// TIA Portal V17 export
// export: Created 2026-04-12T10:31:28.5302505Z, ExportSetting WithDefaults, DisplayName Totally Integrated Automation Portal, DisplayVersion V17 Update 4, DisplayName TIA Portal Openness, DisplayVersion V17 Update 4, DisplayName TIA Portal Version Control Interface, DisplayVersion V17, DisplayName SINAMICS Startdrive Advanced, DisplayVersion V17, DisplayName SINAMICS Startdrive G130, G150, S120, S150, SINAMICS MV, S210, DisplayVersion V17, DisplayName SINAMICS Startdrive G110M, G120, G120C, G120D, G120P, G115D, DisplayVersion V17, DisplayName STEP 7 Professional, DisplayVersion V17 Update 4, DisplayName STEP 7 Safety, DisplayVersion V17, DisplayName WinCC Advanced, DisplayVersion V17 Update 4
FUNCTION "设定值传递" : Void   // FC1, LAD
{ S7_Optimized_Access := 'TRUE' }
VERSION : 0.1
// stored: AutoNumber false, IsIECCheckEnabled false, SetENOAutomatically false, UDAEnableTagReadback false
   VAR_TEMP   // added for the SCL form of the ladder/FBD networks
      _w1 : Bool;
      _w2 : Bool;
   END_VAR
BEGIN

REGION Network 1: 程序停止时
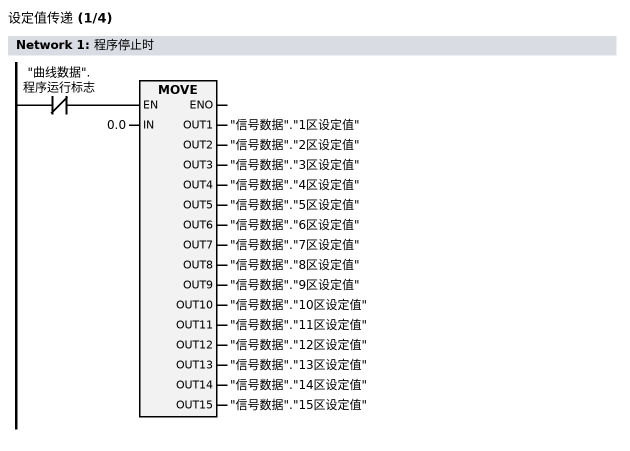
   RUNG wire#powerrail
      I_Contact( "曲线数据".程序运行标志 )
      Move(in := 0.0, out1 => "信号数据"."1区设定值", out2 => "信号数据"."2区设定值", out3 => "信号数据"."3区设定值", out4 => "信号数据"."4区设定值", out5 => "信号数据"."5区设定值", out6 => "信号数据"."6区设定值", out7 => "信号数据"."7区设定值", out8 => "信号数据"."8区设定值", out9 => "信号数据"."9区设定值", out10 => "信号数据"."10区设定值", out11 => "信号数据"."11区设定值", out12 => "信号数据"."12区设定值", out13 => "信号数据"."13区设定值", out14 => "信号数据"."14区设定值", out15 => "信号数据"."15区设定值")
   END_RUNG
   // the same network as SCL:
   IF NOT "曲线数据".程序运行标志 THEN
       "信号数据"."1区设定值" := 0.0;
       "信号数据"."2区设定值" := 0.0;
       "信号数据"."3区设定值" := 0.0;
       "信号数据"."4区设定值" := 0.0;
       "信号数据"."5区设定值" := 0.0;
       "信号数据"."6区设定值" := 0.0;
       "信号数据"."7区设定值" := 0.0;
       "信号数据"."8区设定值" := 0.0;
       "信号数据"."9区设定值" := 0.0;
       "信号数据"."10区设定值" := 0.0;
       "信号数据"."11区设定值" := 0.0;
       "信号数据"."12区设定值" := 0.0;
       "信号数据"."13区设定值" := 0.0;
       "信号数据"."14区设定值" := 0.0;
       "信号数据"."15区设定值" := 0.0;
   END_IF;
END_REGION

REGION Network 2: 程序运行但未暂停时
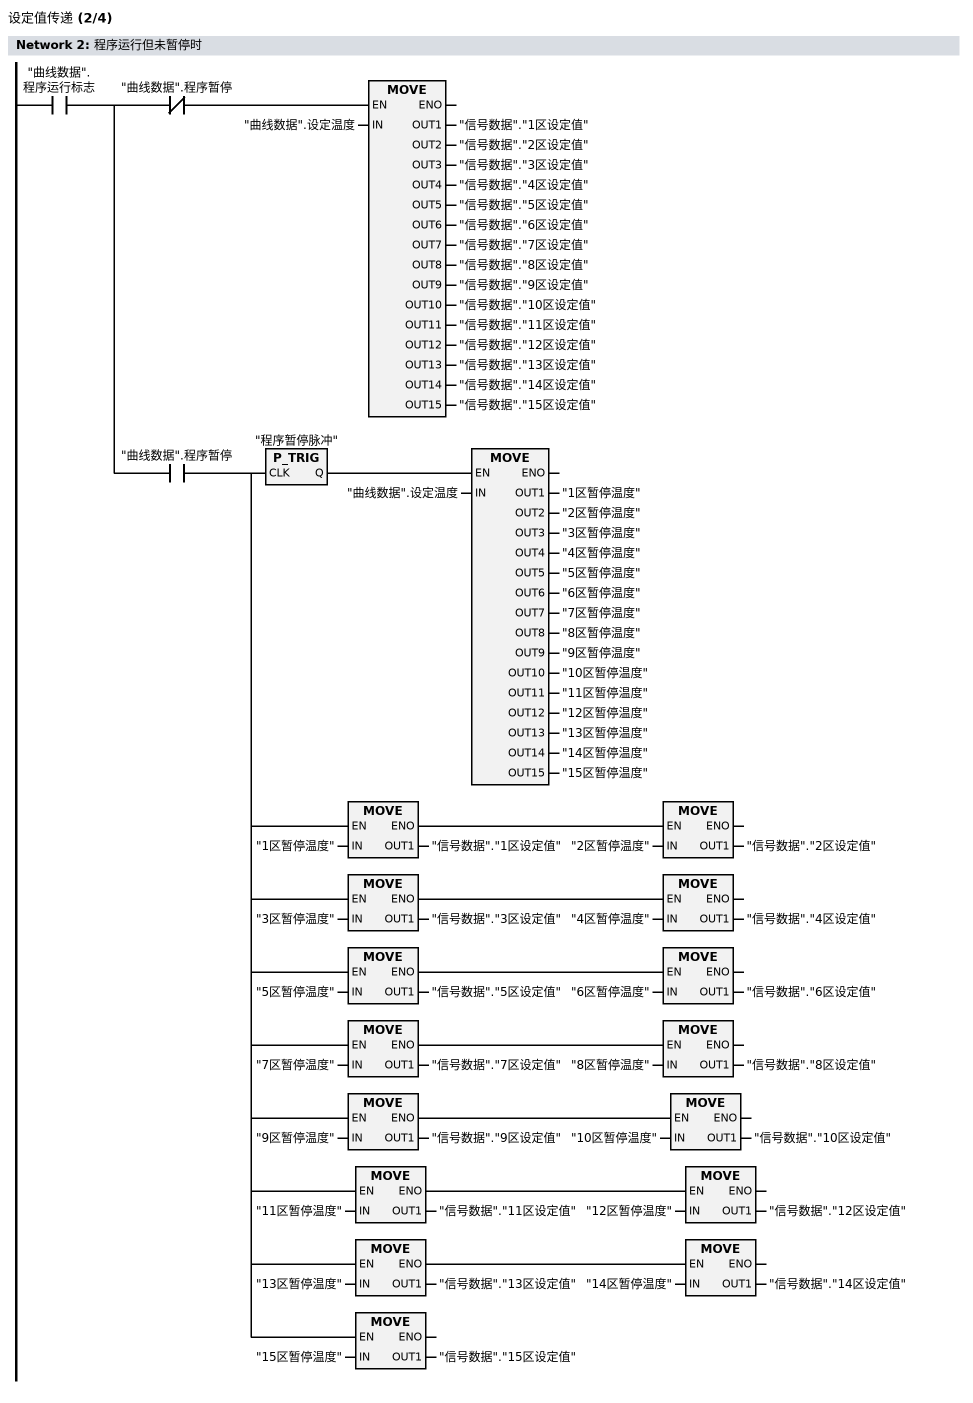
   RUNG wire#powerrail
      Contact( "曲线数据".程序运行标志 )
      wire#w1
      I_Contact( "曲线数据".程序暂停 )
      Move(in := "曲线数据".设定温度, out1 => "信号数据"."1区设定值", out2 => "信号数据"."2区设定值", out3 => "信号数据"."3区设定值", out4 => "信号数据"."4区设定值", out5 => "信号数据"."5区设定值", out6 => "信号数据"."6区设定值", out7 => "信号数据"."7区设定值", out8 => "信号数据"."8区设定值", out9 => "信号数据"."9区设定值", out10 => "信号数据"."10区设定值", out11 => "信号数据"."11区设定值", out12 => "信号数据"."12区设定值", out13 => "信号数据"."13区设定值", out14 => "信号数据"."14区设定值", out15 => "信号数据"."15区设定值")
   END_RUNG
   RUNG wire#w1
      Contact( "曲线数据".程序暂停 )
      wire#w2
      P_Trig( "程序暂停脉冲" )
      Move(in := "曲线数据".设定温度, out1 => "1区暂停温度", out2 => "2区暂停温度", out3 => "3区暂停温度", out4 => "4区暂停温度", out5 => "5区暂停温度", out6 => "6区暂停温度", out7 => "7区暂停温度", out8 => "8区暂停温度", out9 => "9区暂停温度", out10 => "10区暂停温度", out11 => "11区暂停温度", out12 => "12区暂停温度", out13 => "13区暂停温度", out14 => "14区暂停温度", out15 => "15区暂停温度")
   END_RUNG
   RUNG wire#w2
      Move(in := "1区暂停温度", out1 => "信号数据"."1区设定值")
      Move(in := "2区暂停温度", out1 => "信号数据"."2区设定值")
   END_RUNG
   RUNG wire#w2
      Move(in := "3区暂停温度", out1 => "信号数据"."3区设定值")
      Move(in := "4区暂停温度", out1 => "信号数据"."4区设定值")
   END_RUNG
   RUNG wire#w2
      Move(in := "5区暂停温度", out1 => "信号数据"."5区设定值")
      Move(in := "6区暂停温度", out1 => "信号数据"."6区设定值")
   END_RUNG
   RUNG wire#w2
      Move(in := "7区暂停温度", out1 => "信号数据"."7区设定值")
      Move(in := "8区暂停温度", out1 => "信号数据"."8区设定值")
   END_RUNG
   RUNG wire#w2
      Move(in := "9区暂停温度", out1 => "信号数据"."9区设定值")
      Move(in := "10区暂停温度", out1 => "信号数据"."10区设定值")
   END_RUNG
   RUNG wire#w2
      Move(in := "11区暂停温度", out1 => "信号数据"."11区设定值")
      Move(in := "12区暂停温度", out1 => "信号数据"."12区设定值")
   END_RUNG
   RUNG wire#w2
      Move(in := "13区暂停温度", out1 => "信号数据"."13区设定值")
      Move(in := "14区暂停温度", out1 => "信号数据"."14区设定值")
   END_RUNG
   RUNG wire#w2
      Move(in := "15区暂停温度", out1 => "信号数据"."15区设定值")
   END_RUNG
   // the same network as SCL:
   IF "曲线数据".程序运行标志 AND NOT "曲线数据".程序暂停 THEN
       "信号数据"."1区设定值" := "曲线数据".设定温度;
       "信号数据"."2区设定值" := "曲线数据".设定温度;
       "信号数据"."3区设定值" := "曲线数据".设定温度;
       "信号数据"."4区设定值" := "曲线数据".设定温度;
       "信号数据"."5区设定值" := "曲线数据".设定温度;
       "信号数据"."6区设定值" := "曲线数据".设定温度;
       "信号数据"."7区设定值" := "曲线数据".设定温度;
       "信号数据"."8区设定值" := "曲线数据".设定温度;
       "信号数据"."9区设定值" := "曲线数据".设定温度;
       "信号数据"."10区设定值" := "曲线数据".设定温度;
       "信号数据"."11区设定值" := "曲线数据".设定温度;
       "信号数据"."12区设定值" := "曲线数据".设定温度;
       "信号数据"."13区设定值" := "曲线数据".设定温度;
       "信号数据"."14区设定值" := "曲线数据".设定温度;
       "信号数据"."15区设定值" := "曲线数据".设定温度;
   END_IF;
   #_w1 := "曲线数据".程序运行标志 AND "曲线数据".程序暂停;
   #_w2 := #_w1 AND NOT "程序暂停脉冲";   // rising edge
   "程序暂停脉冲" := #_w1;
   IF #_w2 THEN
       "1区暂停温度" := "曲线数据".设定温度;
       "2区暂停温度" := "曲线数据".设定温度;
       "3区暂停温度" := "曲线数据".设定温度;
       "4区暂停温度" := "曲线数据".设定温度;
       "5区暂停温度" := "曲线数据".设定温度;
       "6区暂停温度" := "曲线数据".设定温度;
       "7区暂停温度" := "曲线数据".设定温度;
       "8区暂停温度" := "曲线数据".设定温度;
       "9区暂停温度" := "曲线数据".设定温度;
       "10区暂停温度" := "曲线数据".设定温度;
       "11区暂停温度" := "曲线数据".设定温度;
       "12区暂停温度" := "曲线数据".设定温度;
       "13区暂停温度" := "曲线数据".设定温度;
       "14区暂停温度" := "曲线数据".设定温度;
       "15区暂停温度" := "曲线数据".设定温度;
   END_IF;
   IF #_w1 THEN
       "信号数据"."1区设定值" := "1区暂停温度";
       "信号数据"."2区设定值" := "2区暂停温度";
       "信号数据"."3区设定值" := "3区暂停温度";
       "信号数据"."4区设定值" := "4区暂停温度";
       "信号数据"."5区设定值" := "5区暂停温度";
       "信号数据"."6区设定值" := "6区暂停温度";
       "信号数据"."7区设定值" := "7区暂停温度";
       "信号数据"."8区设定值" := "8区暂停温度";
       "信号数据"."9区设定值" := "9区暂停温度";
       "信号数据"."10区设定值" := "10区暂停温度";
       "信号数据"."11区设定值" := "11区暂停温度";
       "信号数据"."12区设定值" := "12区暂停温度";
       "信号数据"."13区设定值" := "13区暂停温度";
       "信号数据"."14区设定值" := "14区暂停温度";
       "信号数据"."15区设定值" := "15区暂停温度";
   END_IF;
END_REGION

REGION Network 3: 程序运行瞬间复位自动
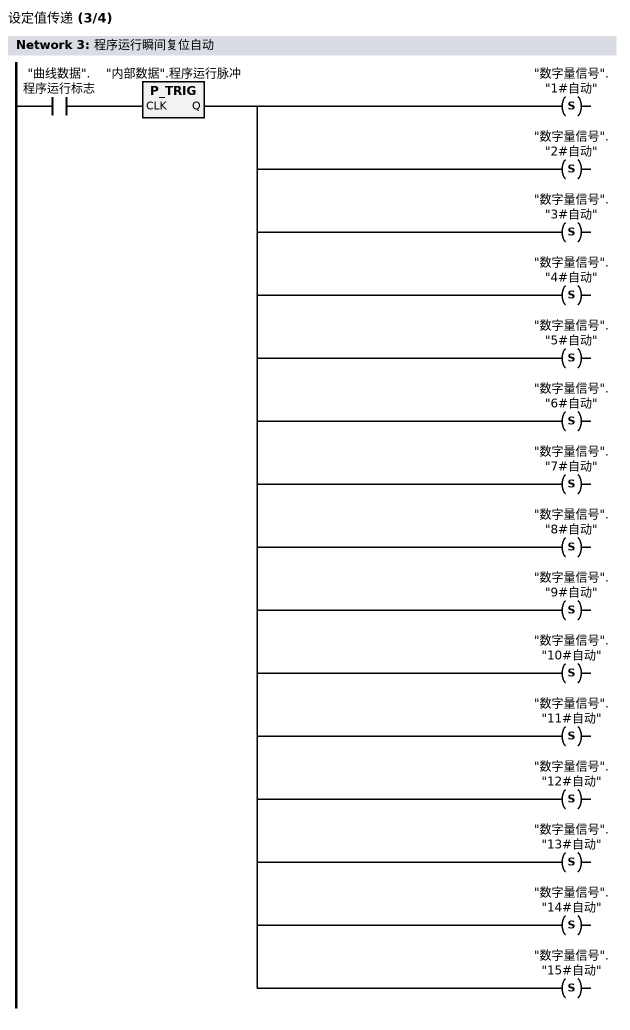
   RUNG wire#powerrail
      Contact( "曲线数据".程序运行标志 )
      P_Trig( "内部数据".程序运行脉冲 )
      wire#w1
      S_Coil( "数字量信号"."1#自动" )
   END_RUNG
   RUNG wire#w1
      S_Coil( "数字量信号"."2#自动" )
   END_RUNG
   RUNG wire#w1
      S_Coil( "数字量信号"."3#自动" )
   END_RUNG
   RUNG wire#w1
      S_Coil( "数字量信号"."4#自动" )
   END_RUNG
   RUNG wire#w1
      S_Coil( "数字量信号"."5#自动" )
   END_RUNG
   RUNG wire#w1
      S_Coil( "数字量信号"."6#自动" )
   END_RUNG
   RUNG wire#w1
      S_Coil( "数字量信号"."7#自动" )
   END_RUNG
   RUNG wire#w1
      S_Coil( "数字量信号"."8#自动" )
   END_RUNG
   RUNG wire#w1
      S_Coil( "数字量信号"."9#自动" )
   END_RUNG
   RUNG wire#w1
      S_Coil( "数字量信号"."10#自动" )
   END_RUNG
   RUNG wire#w1
      S_Coil( "数字量信号"."11#自动" )
   END_RUNG
   RUNG wire#w1
      S_Coil( "数字量信号"."12#自动" )
   END_RUNG
   RUNG wire#w1
      S_Coil( "数字量信号"."13#自动" )
   END_RUNG
   RUNG wire#w1
      S_Coil( "数字量信号"."14#自动" )
   END_RUNG
   RUNG wire#w1
      S_Coil( "数字量信号"."15#自动" )
   END_RUNG
   // the same network as SCL:
   #_w1 := "曲线数据".程序运行标志 AND NOT "内部数据".程序运行脉冲;   // rising edge
   "内部数据".程序运行脉冲 := "曲线数据".程序运行标志;
   IF #_w1 THEN
       "数字量信号"."1#自动" := TRUE;
       "数字量信号"."2#自动" := TRUE;
       "数字量信号"."3#自动" := TRUE;
       "数字量信号"."4#自动" := TRUE;
       "数字量信号"."5#自动" := TRUE;
       "数字量信号"."6#自动" := TRUE;
       "数字量信号"."7#自动" := TRUE;
       "数字量信号"."8#自动" := TRUE;
       "数字量信号"."9#自动" := TRUE;
       "数字量信号"."10#自动" := TRUE;
       "数字量信号"."11#自动" := TRUE;
       "数字量信号"."12#自动" := TRUE;
       "数字量信号"."13#自动" := TRUE;
       "数字量信号"."14#自动" := TRUE;
       "数字量信号"."15#自动" := TRUE;
   END_IF;
END_REGION

REGION Network 4: 当前段斜率
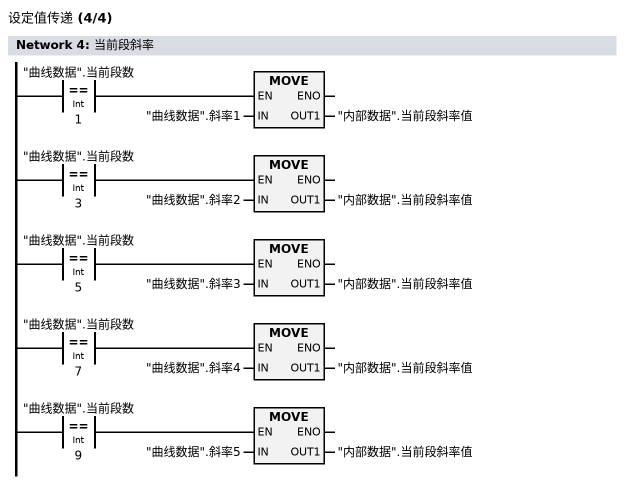
   RUNG wire#powerrail
      { S7_Templates := "SrcType := Int" } EQ_Contact(in1 := "曲线数据".当前段数, in2 := 1)
      Move(in := "曲线数据".斜率1, out1 => "内部数据".当前段斜率值)
   END_RUNG
   RUNG wire#powerrail
      { S7_Templates := "SrcType := Int" } EQ_Contact(in1 := "曲线数据".当前段数, in2 := 3)
      Move(in := "曲线数据".斜率2, out1 => "内部数据".当前段斜率值)
   END_RUNG
   RUNG wire#powerrail
      { S7_Templates := "SrcType := Int" } EQ_Contact(in1 := "曲线数据".当前段数, in2 := 5)
      Move(in := "曲线数据".斜率3, out1 => "内部数据".当前段斜率值)
   END_RUNG
   RUNG wire#powerrail
      { S7_Templates := "SrcType := Int" } EQ_Contact(in1 := "曲线数据".当前段数, in2 := 7)
      Move(in := "曲线数据".斜率4, out1 => "内部数据".当前段斜率值)
   END_RUNG
   RUNG wire#powerrail
      { S7_Templates := "SrcType := Int" } EQ_Contact(in1 := "曲线数据".当前段数, in2 := 9)
      Move(in := "曲线数据".斜率5, out1 => "内部数据".当前段斜率值)
   END_RUNG
   // the same network as SCL:
   IF "曲线数据".当前段数 = 1 THEN "内部数据".当前段斜率值 := "曲线数据".斜率1; END_IF;
   IF "曲线数据".当前段数 = 3 THEN "内部数据".当前段斜率值 := "曲线数据".斜率2; END_IF;
   IF "曲线数据".当前段数 = 5 THEN "内部数据".当前段斜率值 := "曲线数据".斜率3; END_IF;
   IF "曲线数据".当前段数 = 7 THEN "内部数据".当前段斜率值 := "曲线数据".斜率4; END_IF;
   IF "曲线数据".当前段数 = 9 THEN "内部数据".当前段斜率值 := "曲线数据".斜率5; END_IF;
END_REGION
END_FUNCTION
